// Mitsubishi GX Works2 project: PLC_GROUP7   PLC: FX3G

// global labels: Global1
VAR_GLOBAL
  start_day_button AT X007 : BOOL;
  end_day AT M1 : BOOL;
  start_production AT M2 : BOOL;
  start_day_lamp AT Y007 : BOOL;
  emergency_button AT X011 : BOOL;
  choose_beer_type AT X001 : BOOL;
  Analog_input1 AT D8280 : INT;
END_VAR
VAR_GLOBAL CONSTANT
  Div_analog1 : INT := 400;
END_VAR
VAR_GLOBAL
  save_beer_type AT D8201 : INT;
  start_cooking_phase AT M6 : BOOL;
  is_beer_cooked AT TC1 : BOOL;
END_VAR
VAR_GLOBAL CONSTANT
  wait_4_sec : INT := 40;
END_VAR
VAR_GLOBAL
  finish_cooking AT TS1 : BOOL;
  cooking_lamp AT Y001 : BOOL;
END_VAR
VAR_GLOBAL CONSTANT
  is_it_plinzer : INT := 6;
  is_it_lagger : INT := 5;
END_VAR
VAR_GLOBAL
  try_make_plinzer_beer AT M7 : BOOL;
  try_make_lagger_beer AT M8 : BOOL;
END_VAR
VAR_GLOBAL CONSTANT
  sub_120 : REAL := 120;
  sub_6 : REAL := 6;
END_VAR
VAR_GLOBAL
  yeat_input AT D1100 : REAL;
  yeast_stock AT D1102 : REAL;
  malt_input AT D1104 : REAL;
  malt_stock AT D1106 : REAL;
  cuscuta_input AT D1108 : REAL;
  cuscuta_stock AT D1110 : REAL;
  insert_before_day_start_stock AT M9 : BOOL;
  start_cooking_beer AT M10 : BOOL;
END_VAR
VAR_GLOBAL CONSTANT
  sub_150 : REAL := 150;
  sub_12 : REAL := 12;
  sub_60 : REAL := 60;
END_VAR
VAR_GLOBAL
  ferment_button AT X005 : BOOL;
  ezer_for_blinking_light AT M0 : BOOL;
  Blink_light_y3 AT TC3 : BOOL;
END_VAR
VAR_GLOBAL CONSTANT
  counter_blink_y3 : INT := 5;
END_VAR
VAR_GLOBAL
  stop_blink_y3 AT TS3 : BOOL;
  light_lamp_y3 AT Y003 : BOOL;
  Blink_light_y4 AT TC4 : BOOL;
END_VAR
VAR_GLOBAL CONSTANT
  counter_blink_y4 : INT := 5;
END_VAR
VAR_GLOBAL
  stop_blink_y4 AT TS4 : BOOL;
  light_lamp_y4 AT Y004 : BOOL;
  timer_blinking_plinzer AT TC5 : BOOL;
END_VAR
VAR_GLOBAL CONSTANT
  conuter_blink_4 : INT := 40;
END_VAR
VAR_GLOBAL
  stop_ferment AT TS5 : BOOL;
  beer_storage AT D1112 : REAL;
  finish_plinzer_ferment AT M11 : BOOL;
  finish_lagger_ferment AT M12 : BOOL;
  timer_blinking_lagger AT TC6 : BOOL;
END_VAR
VAR_GLOBAL CONSTANT
  counter_blink_3 : INT := 30;
END_VAR
VAR_GLOBAL
  stop_lagger_ferment AT TS6 : BOOL;
  stop_plinzer_ferment AT TS5 : BOOL;
  start_storing_beer_button AT X002 : BOOL;
  insert_beer_to_storage AT X000 : BOOL;
  count_beer_in_store AT CC1 : BOOL;
END_VAR
VAR_GLOBAL CONSTANT
  counter_6 : INT := 6;
END_VAR
VAR_GLOBAL
  finish_storing_beers AT CS1 : BOOL;
  Beer_storing_lamp AT Y002 : BOOL;
END_VAR
VAR_GLOBAL CONSTANT
  Add_1 : REAL := 1;
  Div_analog2 : REAL := 40;
END_VAR
VAR_GLOBAL
  num_of_beer_packs AT D1114 : REAL;
  Analog_Output AT D8282 : INT;
END_VAR
VAR_GLOBAL CONSTANT
  min_yeast : REAL := 120;
  mmin_malt : REAL := 6;
  min_cuscuta : REAL := 54;
END_VAR
VAR_GLOBAL
  out_of_stock AT M3 : BOOL;
  check_all_button_closed AT M13 : BOOL;
  cant_produce_plinzer AT M13 : BOOL;
END_VAR
VAR_GLOBAL CONSTANT
  min_lagger_yeast : REAL := 150;
  min_lagger_malt : REAL := 12;
  min_lagger_cuscuta : REAL := 60;
END_VAR
VAR_GLOBAL
  cant_produce_lagger AT M14 : BOOL;
  reset_day AT M15 : BOOL;
  ezer_for_starting_new_day AT M16 : BOOL;
END_VAR
VAR_GLOBAL CONSTANT
  sub_54 : REAL := 54;
END_VAR
VAR_GLOBAL
  add_to_cooking_storage_lamp AT M17 : BOOL;
END_VAR
VAR_GLOBAL CONSTANT
  Add_180 : REAL := 180;
END_VAR
VAR_GLOBAL
  cooking_storeage AT D1116 : REAL;
END_VAR
VAR_GLOBAL CONSTANT
  Add_222 : REAL := 222;
END_VAR
VAR_GLOBAL
  ferment_storage AT D1118 : REAL;
  add_to_cooking_lagger AT M18 : BOOL;
END_VAR

// task Task_01 (event TRUE, interval 0, priority 31): POU_01

PROGRAM POU_01
(* structured ladder/FBD written out as ST: instructions are called as NAME(EN, inputs, outputs); _pN, _eN, _tN stand for wires *)
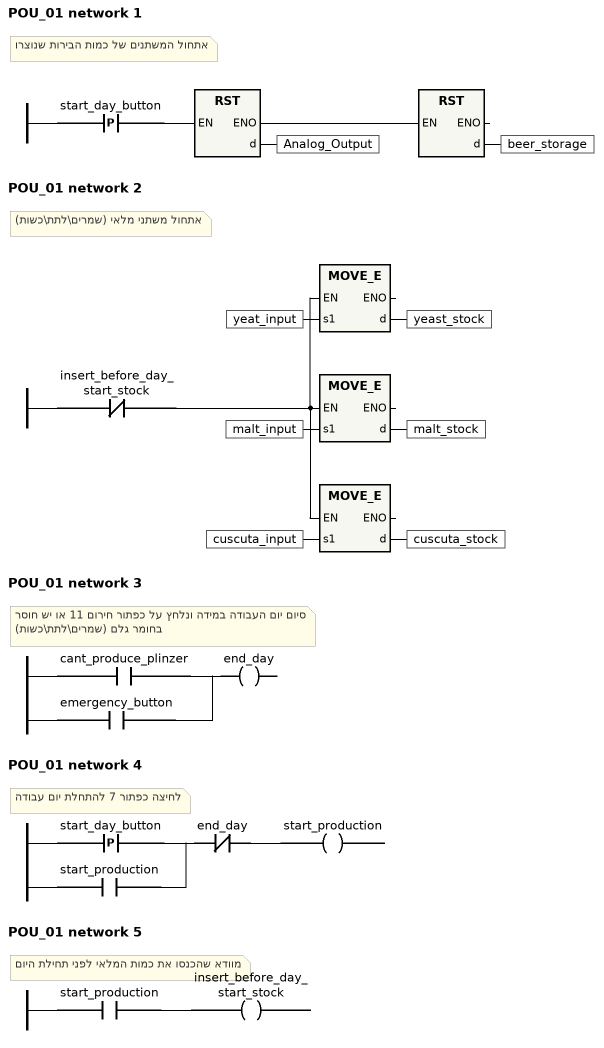
(* network 1 *)
(* אתחול המשתנים של כמות הבירות שנוצרו *)
_e1 := RST(LDP(TRUE, start_day_button), Analog_Output);
RST(_e1, beer_storage);
(* network 2 *)
(* אתחול משתני מלאי (שמרים\לתת\כשות) *)
_p1 := NOT insert_before_day_start_stock;
MOVE_E(_p1, yeat_input, yeast_stock);
MOVE_E(_p1, malt_input, malt_stock);
MOVE_E(_p1, cuscuta_input, cuscuta_stock);
(* network 3 *)
(* סיום יום העבודה במידה ונלחץ על כפתור חירום 11 או יש חוסר בחומר גלם (שמרים\לתת\כשות) *)
end_day := cant_produce_plinzer OR emergency_button;
(* network 4 *)
(* לחיצה כפתור 7 להתחלת יום עבודה *)
start_production := (LDP(TRUE, start_day_button) OR start_production) AND NOT end_day;
(* network 5 *)
(* מוודא שהכנסו את כמות המלאי לפני תחילת היום *)
insert_before_day_start_stock := start_production;
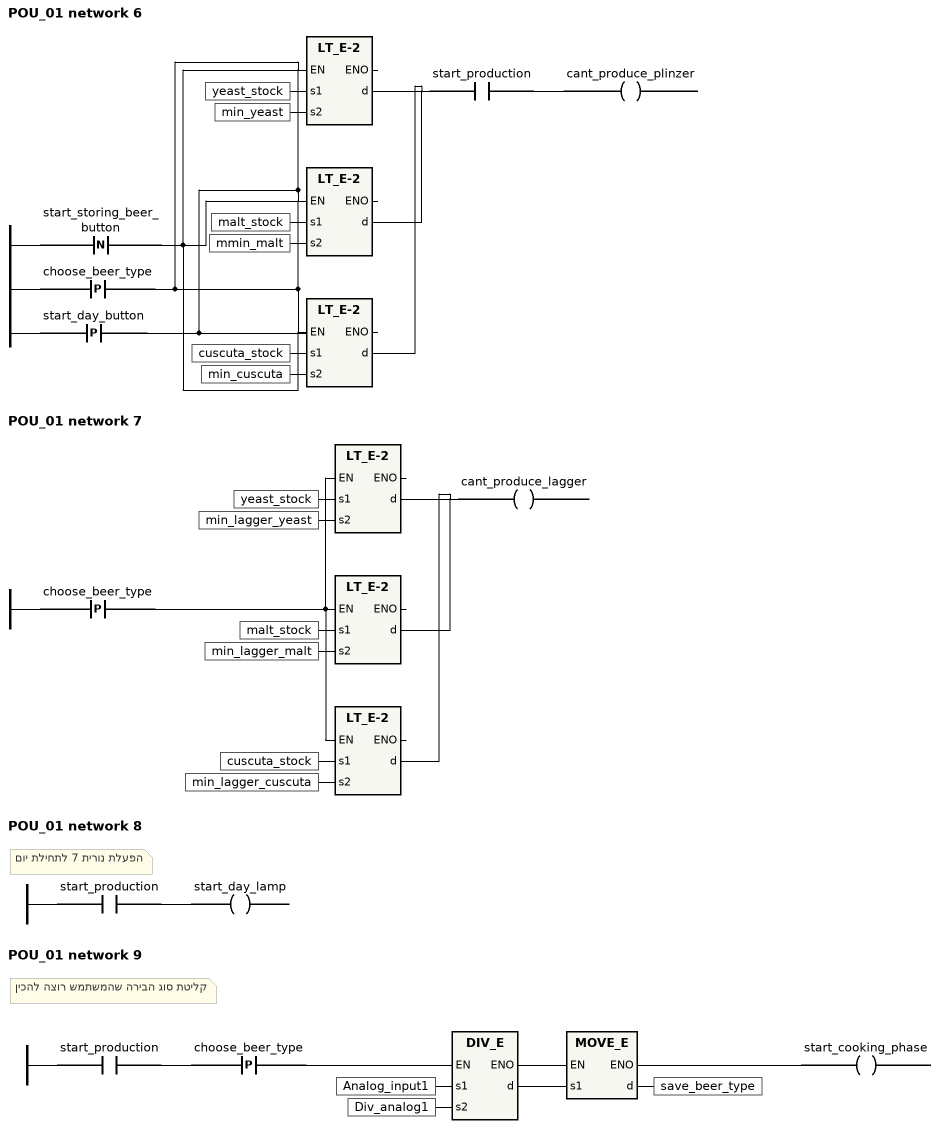
(* network 6 *)
_p1 := LDF(TRUE, start_storing_beer_button) OR LDP(TRUE, choose_beer_type) OR LDP(TRUE, start_day_button);
LT_E(_p1, yeast_stock, min_yeast, _t2);
LT_E(_p1, malt_stock, mmin_malt, _t3);
LT_E(_p1, cuscuta_stock, min_cuscuta, _t4);
cant_produce_plinzer := (_t2 OR _t3 OR _t4) AND start_production;
(* network 7 *)
_p1 := LDP(TRUE, choose_beer_type);
LT_E(_p1, yeast_stock, min_lagger_yeast, _t2);
LT_E(_p1, malt_stock, min_lagger_malt, _t3);
LT_E(_p1, cuscuta_stock, min_lagger_cuscuta, _t4);
cant_produce_lagger := _t2 OR _t3 OR _t4;
(* network 8 *)
(* הפעלת נורית 7 לתחילת יום *)
start_day_lamp := start_production;
(* network 9 *)
(* קליטת סוג הבירה שהמשתמש רוצה להכין *)
_e2 := DIV_E(start_production AND LDP(TRUE, choose_beer_type), Analog_input1, Div_analog1, _t1);
_e3 := MOVE_E(_e2, _t1, save_beer_type);
start_cooking_phase := _e3;
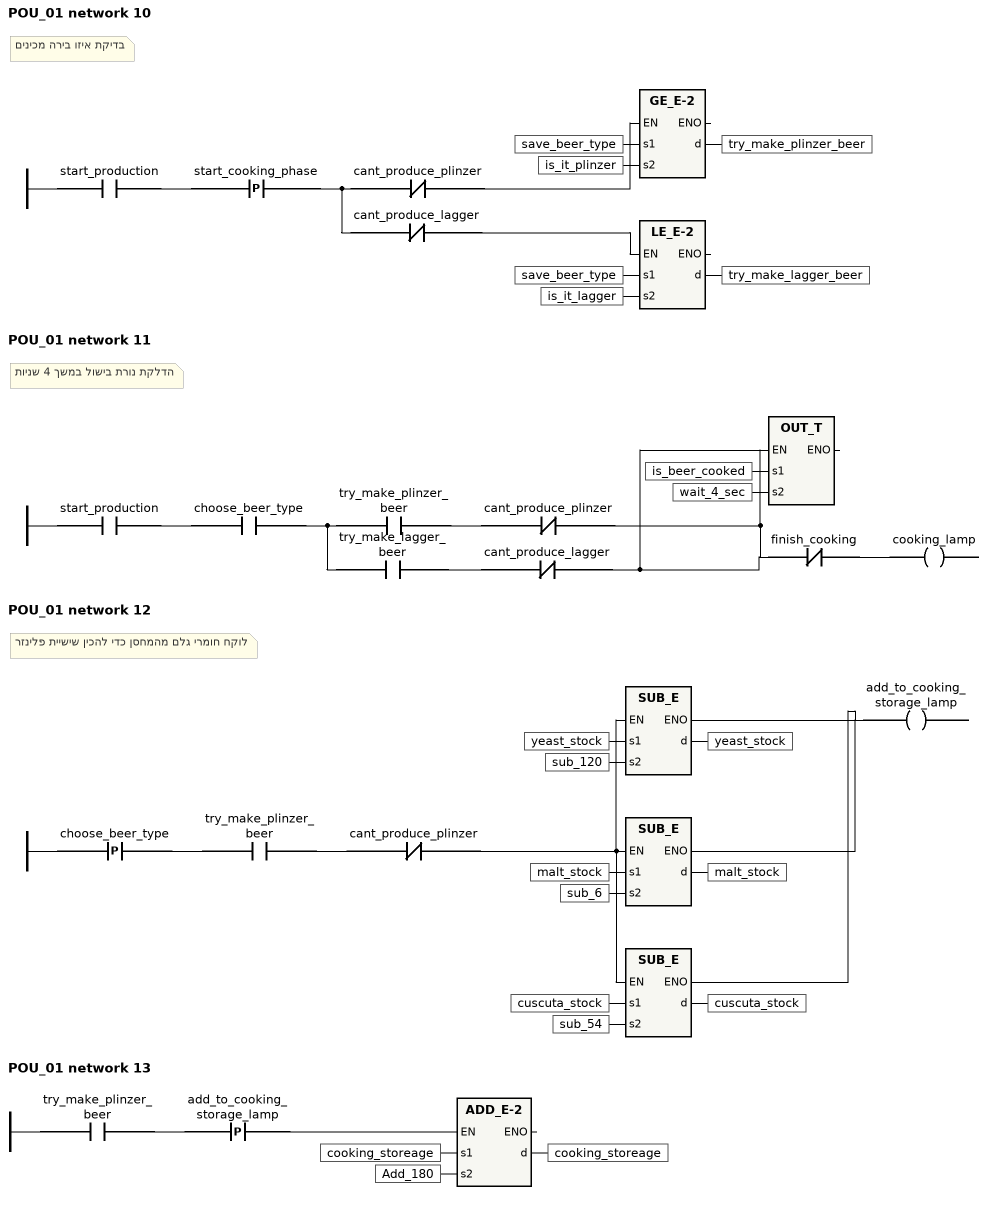
(* network 10 *)
(* בדיקת איזו בירה מכינים *)
_p1 := start_production AND LDP(TRUE, start_cooking_phase);
GE_E(_p1 AND NOT cant_produce_plinzer, save_beer_type, is_it_plinzer, try_make_plinzer_beer);
LE_E(_p1 AND NOT cant_produce_lagger, save_beer_type, is_it_lagger, try_make_lagger_beer);
(* network 11 *)
(* הדלקת נורת בישול במשך 4 שניות *)
_p1 := start_production AND choose_beer_type;
_p2 := (_p1 AND try_make_plinzer_beer AND NOT cant_produce_plinzer) OR (_p1 AND try_make_lagger_beer AND NOT cant_produce_lagger);
OUT_T(_p2, is_beer_cooked, wait_4_sec);
cooking_lamp := _p2 AND NOT finish_cooking;
(* network 12 *)
(* לוקח חומרי גלם מהמחסן כדי להכין שישיית פלינזר *)
_p1 := LDP(TRUE, choose_beer_type) AND try_make_plinzer_beer AND NOT cant_produce_plinzer;
_e2 := SUB_E(_p1, yeast_stock, sub_120, yeast_stock);
_e3 := SUB_E(_p1, malt_stock, sub_6, malt_stock);
_e4 := SUB_E(_p1, cuscuta_stock, sub_54, cuscuta_stock);
add_to_cooking_storage_lamp := _e2 OR _e3 OR _e4;
(* network 13 *)
ADD_E(try_make_plinzer_beer AND LDP(TRUE, add_to_cooking_storage_lamp), cooking_storeage, Add_180, cooking_storeage);
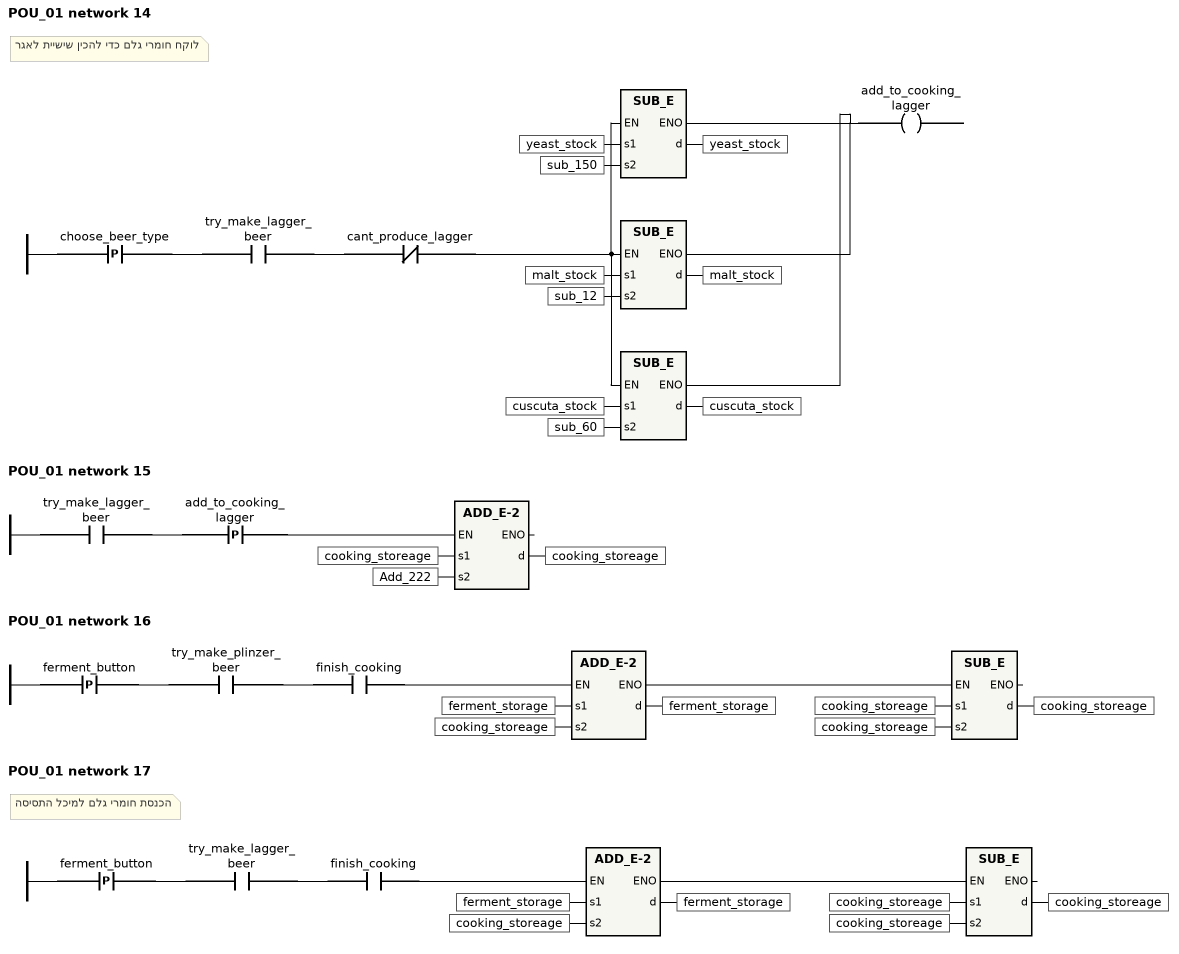
(* network 14 *)
(* לוקח חומרי גלם כדי להכין שישיית לאגר *)
_p1 := LDP(TRUE, choose_beer_type) AND try_make_lagger_beer AND NOT cant_produce_lagger;
_e2 := SUB_E(_p1, yeast_stock, sub_150, yeast_stock);
_e3 := SUB_E(_p1, malt_stock, sub_12, malt_stock);
_e4 := SUB_E(_p1, cuscuta_stock, sub_60, cuscuta_stock);
add_to_cooking_lagger := _e2 OR _e3 OR _e4;
(* network 15 *)
ADD_E(try_make_lagger_beer AND LDP(TRUE, add_to_cooking_lagger), cooking_storeage, Add_222, cooking_storeage);
(* network 16 *)
_e1 := ADD_E(LDP(TRUE, ferment_button) AND try_make_plinzer_beer AND finish_cooking, ferment_storage, cooking_storeage, ferment_storage);
SUB_E(_e1, cooking_storeage, cooking_storeage, cooking_storeage);
(* network 17 *)
(* הכנסת חומרי גלם למיכל התסיסה *)
_e1 := ADD_E(LDP(TRUE, ferment_button) AND try_make_lagger_beer AND finish_cooking, ferment_storage, cooking_storeage, ferment_storage);
SUB_E(_e1, cooking_storeage, cooking_storeage, cooking_storeage);
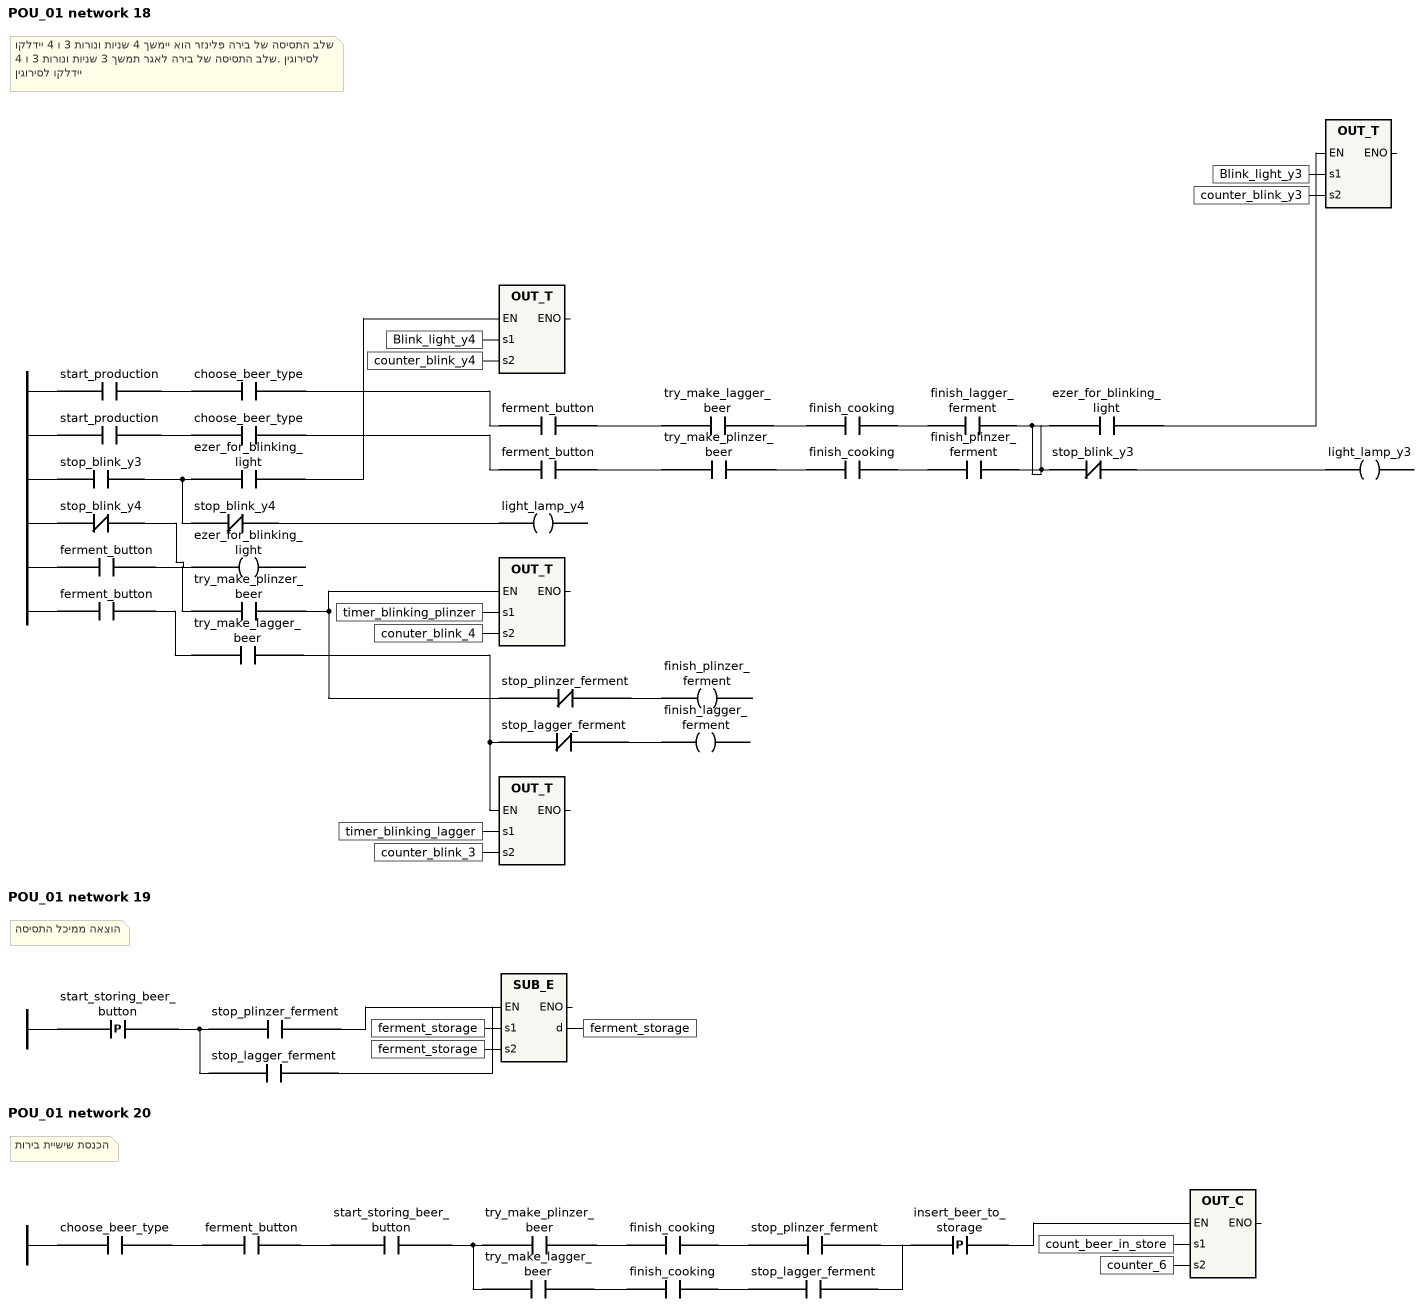
(* network 18 *)
(* שלב התסיסה של בירה פלינזר הוא יימשך 4 שניות ונורות 3 ו 4 יידלקו לסירוגין .שלב התסיסה של בירה לאגר תמשך 3 שניות ונורות 3 ו 4 יידלקו לסירוגין *)
_p1 := (start_production AND choose_beer_type AND ferment_button AND try_make_lagger_beer AND finish_cooking AND finish_lagger_ferment) OR (start_production AND choose_beer_type AND ferment_button AND try_make_plinzer_beer AND finish_cooking AND finish_plinzer_ferment);
OUT_T(_p1 AND ezer_for_blinking_light, Blink_light_y3, counter_blink_y3);
light_lamp_y3 := _p1 AND NOT stop_blink_y3;
OUT_T(stop_blink_y3 AND ezer_for_blinking_light, Blink_light_y4, counter_blink_y4);
light_lamp_y4 := stop_blink_y3 AND NOT stop_blink_y4;
ezer_for_blinking_light := NOT stop_blink_y4;
_p2 := ferment_button AND try_make_plinzer_beer;
OUT_T(_p2, timer_blinking_plinzer, conuter_blink_4);
finish_plinzer_ferment := _p2 AND NOT stop_plinzer_ferment;
_p3 := ferment_button AND try_make_lagger_beer;
OUT_T(_p3, timer_blinking_lagger, counter_blink_3);
finish_lagger_ferment := _p3 AND NOT stop_lagger_ferment;
(* network 19 *)
(* הוצאה ממיכל התסיסה *)
_p1 := LDP(TRUE, start_storing_beer_button);
SUB_E((_p1 AND stop_plinzer_ferment) OR (_p1 AND stop_lagger_ferment), ferment_storage, ferment_storage, ferment_storage);
(* network 20 *)
(* הכנסת שישיית בירות *)
_p1 := choose_beer_type AND ferment_button AND start_storing_beer_button;
OUT_C(((_p1 AND try_make_plinzer_beer AND finish_cooking AND stop_plinzer_ferment) OR (_p1 AND try_make_lagger_beer AND finish_cooking AND stop_lagger_ferment)) AND LDP(TRUE, insert_beer_to_storage), count_beer_in_store, counter_6);
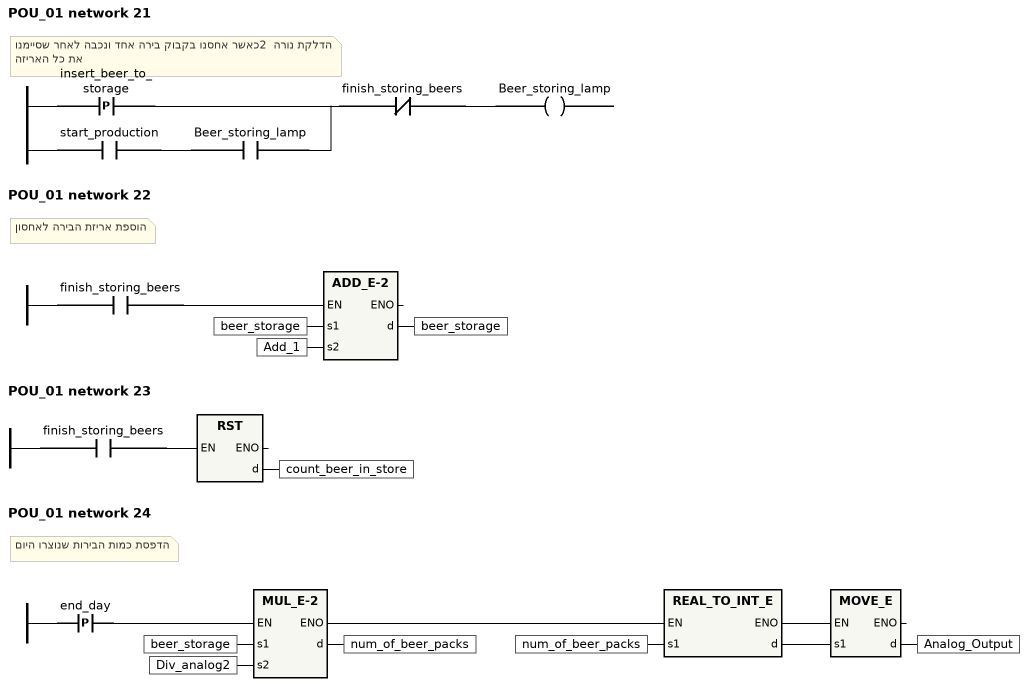
(* network 21 *)
(* הדלקת נורה  2כאשר אחסנו בקבוק בירה אחד ונכבה לאחר שסיימנו את כל האריזה *)
Beer_storing_lamp := (LDP(TRUE, insert_beer_to_storage) OR (start_production AND Beer_storing_lamp)) AND NOT finish_storing_beers;
(* network 22 *)
(* הוספת אריזת הבירה לאחסון *)
ADD_E(finish_storing_beers, beer_storage, Add_1, beer_storage);
(* network 23 *)
RST(finish_storing_beers, count_beer_in_store);
(* network 24 *)
(* הדפסת כמות הבירות שנוצרו היום *)
_e1 := MUL_E(LDP(TRUE, end_day), beer_storage, Div_analog2, num_of_beer_packs);
_e3 := REAL_TO_INT_E(_e1, num_of_beer_packs, _t2);
MOVE_E(_e3, _t2, Analog_Output);
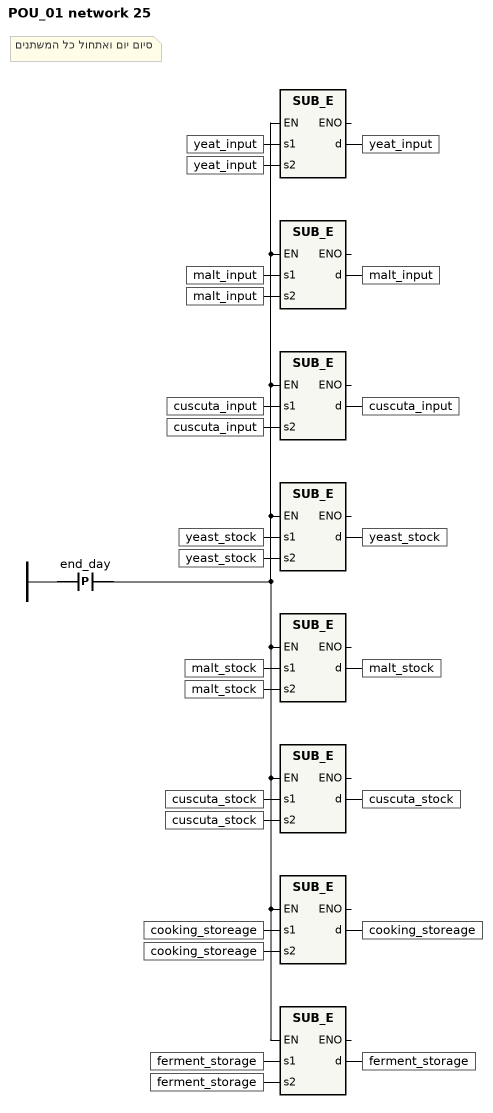
(* network 25 *)
(* סיום יום ואתחול כל המשתנים *)
_p1 := LDP(TRUE, end_day);
SUB_E(_p1, yeat_input, yeat_input, yeat_input);
SUB_E(_p1, malt_input, malt_input, malt_input);
SUB_E(_p1, cuscuta_input, cuscuta_input, cuscuta_input);
SUB_E(_p1, yeast_stock, yeast_stock, yeast_stock);
SUB_E(_p1, malt_stock, malt_stock, malt_stock);
SUB_E(_p1, cuscuta_stock, cuscuta_stock, cuscuta_stock);
SUB_E(_p1, cooking_storeage, cooking_storeage, cooking_storeage);
SUB_E(_p1, ferment_storage, ferment_storage, ferment_storage);
END_PROGRAM
